FUNCTION_BLOCK CROSSCOMM_PEER_24EBE21AE52A465D (* Service Interface Function Block Type *)
  (* Standard: 61499-2 *)
  (* Version 0.0, 9/22/2017, bababen, nxtControl GmbH, template *)
  PACKAGE Main;
  (* Compiler Cpp nxtControl builtin 1.0 *)
  {SET_ATTRIBUTE(Runtime.FBType.ImplementingType, Runtime.System#DYNGEN_CROSSCOMM_PEER)}
  {SET_ATTRIBUTE(Configuration.GenericFBType.InterfaceParams, Runtime.System#<InterfaceList> <EventOutputs> <Event Name="CNF"> <With Var="LExtended" /> <With Var="LRetracted" /> </Event> </EventOutputs> <OutputVars> <VarDeclaration Name="LExtended" Type="BOOL" /> <VarDeclaration Name="LRetracted" Type="BOOL" /> </OutputVars> </InterfaceList>)}
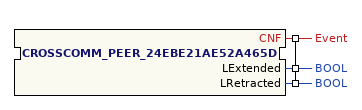
  EVENT_OUTPUT
    CNF WITH LExtended, LRetracted;
  END_EVENT
  VAR_OUTPUT
    LExtended : BOOL;
    LRetracted : BOOL;
  END_VAR
  EC_STATES
    START;
  END_STATES
END_FUNCTION_BLOCK
